// TIA Portal V20 export
DATA_BLOCK "StackToReelCut10"   // DB331
// stored: InstanceOfName typeStackToReelCut, InstanceOfType UDT
"typeStackToReelCut"
   // VAR
   //    Load_Requset : Bool := FALSE;
   //    Load_Busy : Bool := FALSE;
   //    Load_Complete : Bool := FALSE;
   //    Cell_Data_Request : Bool := FALSE;
   //    Cell_Data_Report_Ack : Bool := FALSE;
   //    Cell_Data_Report_Nck : Bool := FALSE;
   //    signal6 : Bool := FALSE;
   //    signal7 : Bool := FALSE;
   //    signal8 : Bool := FALSE;
   //    signal9 : Bool := FALSE;
   //    signal10 : Bool := FALSE;
   //    signal11 : Bool := FALSE;
   //    signal12 : Bool := FALSE;
   //    signal13 : Bool := FALSE;
   //    signal14 : Bool := FALSE;
   //    HeartBeat : Bool := TRUE;
   //    signal16 : Bool := FALSE;
   //    signal17 : Bool := FALSE;
   //    signal18 : Bool := FALSE;
   //    signal19 : Bool := FALSE;
   //    signal20 : Bool := FALSE;
   //    signal21 : Bool := FALSE;
   //    signal22 : Bool := FALSE;
   //    signal23 : Bool := FALSE;
   //    signal24 : Bool := FALSE;
   //    signal25 : Bool := FALSE;
   //    signal26 : Bool := FALSE;
   //    signal27 : Bool := FALSE;
   //    signal28 : Bool := FALSE;
   //    signal29 : Bool := FALSE;
   //    signal30 : Bool := FALSE;
   //    signal31 : Bool := FALSE;
   //    signal32 : Bool := FALSE;
   //    signal33 : Bool := FALSE;
   //    signal34 : Bool := FALSE;
   //    signal35 : Bool := FALSE;
   //    signal36 : Bool := FALSE;
   //    signal37 : Bool := FALSE;
   //    signal38 : Bool := FALSE;
   //    signal39 : Bool := FALSE;
   //    signal40 : Bool := FALSE;
   //    signal41 : Bool := FALSE;
   //    signal42 : Bool := FALSE;
   //    signal43 : Bool := FALSE;
   //    signal44 : Bool := FALSE;
   //    signal45 : Bool := FALSE;
   //    signal46 : Bool := FALSE;
   //    signal47 : Bool := FALSE;
   //    signal48 : Bool := FALSE;
   //    signal49 : Bool := FALSE;
   //    signal50 : Bool := FALSE;
   //    signal51 : Bool := FALSE;
   //    signal52 : Bool := FALSE;
   //    signal53 : Bool := FALSE;
   //    signal54 : Bool := FALSE;
   //    signal55 : Bool := FALSE;
   //    signal56 : Bool := FALSE;
   //    signal57 : Bool := FALSE;
   //    signal58 : Bool := FALSE;
   //    signal59 : Bool := FALSE;
   //    signal60 : Bool := FALSE;
   //    signal61 : Bool := FALSE;
   //    signal62 : Bool := FALSE;
   //    signal63 : Bool := FALSE;
   //    signal64 : Bool := FALSE;
   //    signal65 : Bool := FALSE;
   //    signal66 : Bool := FALSE;
   //    signal67 : Bool := FALSE;
   //    signal68 : Bool := FALSE;
   //    signal69 : Bool := FALSE;
   //    signal70 : Bool := FALSE;
   //    signal71 : Bool := FALSE;
   //    signal72 : Bool := FALSE;
   //    signal73 : Bool := FALSE;
   //    signal74 : Bool := FALSE;
   //    signal75 : Bool := FALSE;
   //    signal76 : Bool := FALSE;
   //    signal77 : Bool := FALSE;
   //    signal78 : Bool := FALSE;
   //    signal79 : Bool := FALSE;
   //    signal80 : Bool := FALSE;
   //    signal81 : Bool := FALSE;
   //    signal82 : Bool := FALSE;
   //    signal83 : Bool := FALSE;
   //    signal84 : Bool := FALSE;
   //    signal85 : Bool := FALSE;
   //    signal86 : Bool := FALSE;
   //    signal87 : Bool := FALSE;
   //    signal88 : Bool := FALSE;
   //    signal89 : Bool := FALSE;
   //    signal90 : Bool := FALSE;
   //    signal91 : Bool := FALSE;
   //    signal92 : Bool := FALSE;
   //    signal93 : Bool := FALSE;
   //    signal94 : Bool := FALSE;
   //    signal95 : Bool := FALSE;
   // END_VAR
BEGIN
END_DATA_BLOCK
